// TIA Portal V17 export
// export: Created 2024-09-02T12:50:19.4027294Z, ExportSetting WithDefaults, DisplayName Totally Integrated Automation Portal, DisplayVersion V17, DisplayName TIA Portal Openness, DisplayVersion V17, DisplayName TIA Portal Version Control Interface, DisplayVersion V17, DisplayName STEP 7 Professional, DisplayVersion V17, DisplayName STEP 7 Safety, DisplayVersion V17, DisplayName WinCC Professional, DisplayVersion V17
DATA_BLOCK "AnwDB_Desoutter_OP70_2"   // DB110
{ S7_Optimized_Access := 'TRUE'; DB_Accessible_From_OPC_UA := 'FALSE' }
VERSION : 0.1
// stored: AutoNumber false, DBAccessibleFromOPCUA false, IsOnlyStoredInLoadMemory false, IsRetainMemResEnabled false, IsWriteProtectedInAS false, MemoryReserve 0
   VAR
      HMI : Struct
         Visu : Struct
            Output { S7_SetPoint := 'True'} : "Desoutter_Output";
            Input { S7_SetPoint := 'True'} : "Desoutter_Input";
            Temp : Struct
               EchoSelected : Array[0..7] of Bool;
               Select : Array[0..7] of Bool;
            END_STRUCT;
         END_STRUCT;
         Button : Struct
            Reset : Struct
               appearance : Int;
               active : Bool;
            END_STRUCT;
            Start : Struct
               appearance : Int;
               active : Bool;
            END_STRUCT;
            Start_Unscrewing : Struct
               appearance : Int;
               active : Bool;
            END_STRUCT;
            EnblFnc : Int;
            Prg_Nr : Int;
         END_STRUCT;
         Variant_Number : String;
      END_STRUCT;
      ID_of_HCU : String;
      No_Part : Array[1..32] of Char;
      Data_From_Proces1 : Struct
         Torque : Real;
         Angle : Real;
      END_STRUCT;
      Empty_Proces_Data : Struct
         Torque : Real;
         Angle : Real;
      END_STRUCT;
   END_VAR
BEGIN
   No_Part[1..32] := ' ';
END_DATA_BLOCK
